(* CODESYS project e!C_ScaleAnalogIO_Test_1.ecp

Project tree, tasks and I/O mapping:
  Device : 750-8202 PFC200 2ETH RS, WAGO, order no. 0750-8202, version 5.11.1.16
    application Application
      libraries: Util, * (System)
      task Test (cyclic, interval T#50ms, priority 11) calls PLC_PRG
      Data types/
      Global Variables/
        global variables Global_Constants
        global variables Global_Retains
        global variables Global_Variables
        global variables Variable_Configuration
      POUs/
        Diagnostic/
          program ModuleDiagnostic [ST]: ModuleDiagList
        Scaling/
          function block fbScale_AI_455 [ST]
          function block fbScale_AI_457 [ST]
          function block fbScale_AI_457_Positiv [ST]
          function block fbScale_AI_460 [ST]
          function block fbScale_AI_461 [ST]
          function block fbScale_AI_466 [ST]
          function block fbScale_AI_473 [ST]
          function block fbScale_AO_552 [ST]
          function block fbScale_AO_555 [ST]
          function block fbScale_AO_556 [ST]
          function block fbScale_AO_559 [ST]
        program PLC_PRG [CFC]: AnalogInput, AnalogOutput
      Visualizations/
      global variables PersistentVars
      trace Sampling_Trace (task ): 
    DeviceAdapter
    Kbus : Kbus, WAGO, version 1.4.0.2
        unmapped channels: K-BUS diagnostics
    MODBUS
      MODBUS : MODBUS, WAGO, order no. n/a, version 1.1.1.15
    Serial
      COM1 : COM1, WAGO, version 0.0.0.19
  GlobalImagePool
*)

// Device/Application/Global Variables/Global_Constants
VAR_GLOBAL CONSTANT

	LIM_OF_DIAG_MODULES : INT := 100;
	LIM_OF_DIAG_CHANNELS : INT := 8;
	MODULE_DIAG_UNDERRANGE : INT := 16#41;
	MODULE_DIAG_OVERRANGE : INT := 16#42;
	MODULE_DIAG_MSG_UNDERRANGE : STRING(15) := 'Underrange';
	MODULE_DIAG_MSG_OVERRANGE : STRING(15) := 'Overrange';
	MODULE_DIAG_MSG_OK : STRING(15) := 'Ok';

END_VAR

// Device/Application/Global Variables/Global_Retains
VAR_GLOBAL RETAIN

	awDiagDataCapture				: ARRAY[1..LIM_OF_DIAG_MODULES, 1..LIM_OF_DIAG_CHANNELS] OF WORD;

END_VAR

// Device/Application/Global Variables/Global_Variables
VAR_GLOBAL

	asModuleDiag				: ARRAY[1..LIM_OF_DIAG_MODULES, 1..LIM_OF_DIAG_CHANNELS] OF STRING(15);

END_VAR

// Device/Application/Global Variables/Variable_Configuration
VAR_CONFIG
END_VAR

// Device/Application/PersistentVars
VAR_GLOBAL PERSISTENT RETAIN
END_VAR

// Device/Application/POUs/PLC_PRG
PROGRAM PLC_PRG
VAR

	Scale_AI_Pressure_1: fbScale_AI_455;
	Scale_AI_Distance_1: fbScale_AI_473;
	Scale_AI_Level_1: fbScale_AI_466;
	Scale_AI_Temp_1: fbScale_AI_460;
	Scale_AI_EngineTemp_1: fbScale_AI_461;
	Scale_AI_SpeedActual_1: fbScale_AI_457_Positiv;
	Scale_AO_SpeedSet_1: fbScale_AO_559;
	Scale_AO_PressureSet_1: fbScale_AO_555;
	Scale_AO_LevelSet_1: fbScale_AO_556;
	Scale_AO_DistanceSet_1: fbScale_AO_552;

	AI_Pressure_1_Signal: REAL;
	AI_Pressure_1_SignalStatus : BYTE;
	AI_Distance_1_Signal: REAL;
	AI_Distance_1_SignalStatus : BYTE;
	AI_Level_1_Signal: REAL;
	AI_Level_1_SignalStatus : BYTE;
	AI_Temp_1_Signal: REAL;
	AI_Temp_1_SignalStatus : BYTE;
	AI_EngineTemp_1_Signal: REAL;
	AI_EngineTemp_1_SignalStatus : BYTE;
	AI_SpeedActual_1_Signal: REAL;
	AI_SpeedActual_1_SignalStatus: BYTE;
	AO_SpeedSet_1_Signal: REAL;
	AO_SpeedSet_1_SignalStatus: BYTE;
	AO_PressureSet_1_Signal: REAL;
	AO_PressureSet_1_SignalStatus: BYTE;
	AO_LevelSet_1_Signal: REAL;
	AO_LevelSet_1_SignalStatus: BYTE;
	AO_DistanceSet_1_Signal: REAL;
	AO_DistanceSet_1_SignalStatus: BYTE;

	AI_455_1_1_sim: WORD;
	AI_473_1_1_sim: WORD;
	AI_466_1_1_sim: WORD;
	AI_460_1_1_sim: INT;
	AI_461_1_1_sim: INT;
	AI_457_1_1_sim: WORD;
	AO_559_1_1_sim: WORD;
	AO_552_1_1_sim: WORD;
	AO_555_1_1_sim: WORD;
	AO_556_1_1_sim: WORD;

END_VAR

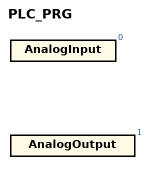
AnalogInput();
AnalogOutput();

ACTION AnalogInput:
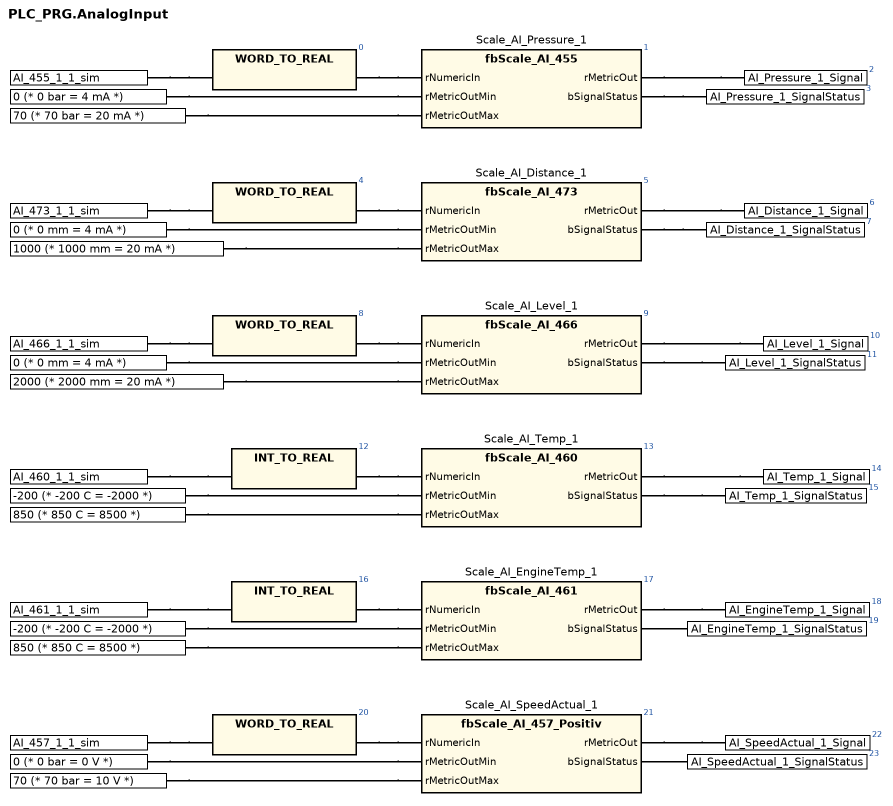
Scale_AI_Pressure_1(
    rNumericIn := WORD_TO_REAL(AI_455_1_1_sim),
    rMetricOutMin := 0 (* 0 bar = 4 mA *),
    rMetricOutMax := 70 (* 70 bar = 20 mA *)); // fbScale_AI_455
AI_Pressure_1_Signal := Scale_AI_Pressure_1.rMetricOut;
AI_Pressure_1_SignalStatus := Scale_AI_Pressure_1.bSignalStatus;
Scale_AI_Distance_1(
    rNumericIn := WORD_TO_REAL(AI_473_1_1_sim),
    rMetricOutMin := 0 (* 0 mm = 4 mA *),
    rMetricOutMax := 1000 (* 1000 mm = 20 mA *)); // fbScale_AI_473
AI_Distance_1_Signal := Scale_AI_Distance_1.rMetricOut;
AI_Distance_1_SignalStatus := Scale_AI_Distance_1.bSignalStatus;
Scale_AI_Level_1(
    rNumericIn := WORD_TO_REAL(AI_466_1_1_sim),
    rMetricOutMin := 0 (* 0 mm = 4 mA *),
    rMetricOutMax := 2000 (* 2000 mm = 20 mA *)); // fbScale_AI_466
AI_Level_1_Signal := Scale_AI_Level_1.rMetricOut;
AI_Level_1_SignalStatus := Scale_AI_Level_1.bSignalStatus;
Scale_AI_Temp_1(
    rNumericIn := INT_TO_REAL(AI_460_1_1_sim),
    rMetricOutMin := -200 (* -200 C = -2000 *),
    rMetricOutMax := 850 (* 850 C = 8500 *)); // fbScale_AI_460
AI_Temp_1_Signal := Scale_AI_Temp_1.rMetricOut;
AI_Temp_1_SignalStatus := Scale_AI_Temp_1.bSignalStatus;
Scale_AI_EngineTemp_1(
    rNumericIn := INT_TO_REAL(AI_461_1_1_sim),
    rMetricOutMin := -200 (* -200 C = -2000 *),
    rMetricOutMax := 850 (* 850 C = 8500 *)); // fbScale_AI_461
AI_EngineTemp_1_Signal := Scale_AI_EngineTemp_1.rMetricOut;
AI_EngineTemp_1_SignalStatus := Scale_AI_EngineTemp_1.bSignalStatus;
Scale_AI_SpeedActual_1(
    rNumericIn := WORD_TO_REAL(AI_457_1_1_sim),
    rMetricOutMin := 0 (* 0 bar = 0 V *),
    rMetricOutMax := 70 (* 70 bar = 10 V *)); // fbScale_AI_457_Positiv
AI_SpeedActual_1_Signal := Scale_AI_SpeedActual_1.rMetricOut;
AI_SpeedActual_1_SignalStatus := Scale_AI_SpeedActual_1.bSignalStatus;
END_ACTION

ACTION AnalogOutput:
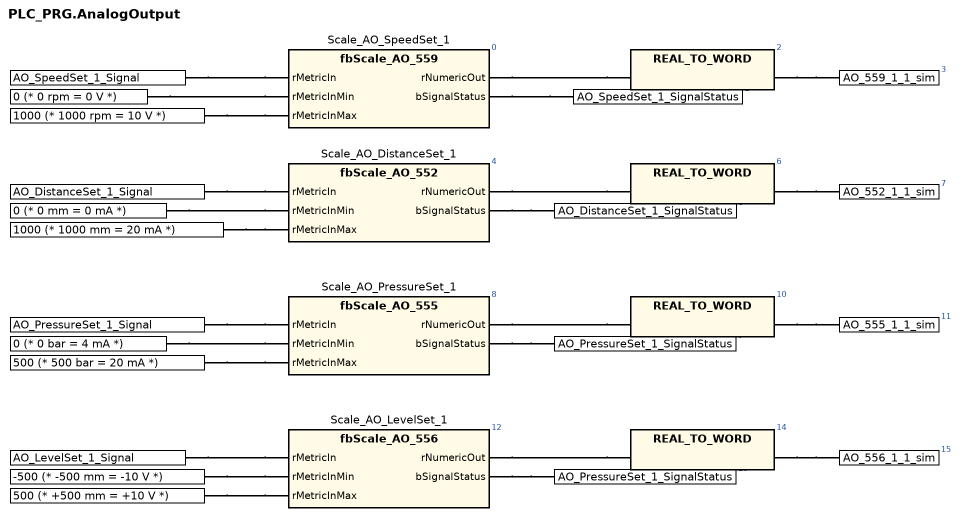
Scale_AO_SpeedSet_1(
    rMetricIn := AO_SpeedSet_1_Signal,
    rMetricInMin := 0 (* 0 rpm = 0 V *),
    rMetricInMax := 1000 (* 1000 rpm = 10 V *)); // fbScale_AO_559
AO_SpeedSet_1_SignalStatus := Scale_AO_SpeedSet_1.bSignalStatus;
AO_559_1_1_sim := REAL_TO_WORD(Scale_AO_SpeedSet_1.rNumericOut);
Scale_AO_DistanceSet_1(
    rMetricIn := AO_DistanceSet_1_Signal,
    rMetricInMin := 0 (* 0 mm = 0 mA *),
    rMetricInMax := 1000 (* 1000 mm = 20 mA *)); // fbScale_AO_552
AO_DistanceSet_1_SignalStatus := Scale_AO_DistanceSet_1.bSignalStatus;
AO_552_1_1_sim := REAL_TO_WORD(Scale_AO_DistanceSet_1.rNumericOut);
Scale_AO_PressureSet_1(
    rMetricIn := AO_PressureSet_1_Signal,
    rMetricInMin := 0 (* 0 bar = 4 mA *),
    rMetricInMax := 500 (* 500 bar = 20 mA *)); // fbScale_AO_555
AO_PressureSet_1_SignalStatus := Scale_AO_PressureSet_1.bSignalStatus;
AO_555_1_1_sim := REAL_TO_WORD(Scale_AO_PressureSet_1.rNumericOut);
Scale_AO_LevelSet_1(
    rMetricIn := AO_LevelSet_1_Signal,
    rMetricInMin := -500 (* -500 mm = -10 V *),
    rMetricInMax := 500 (* +500 mm = +10 V *)); // fbScale_AO_556
AO_PressureSet_1_SignalStatus := Scale_AO_LevelSet_1.bSignalStatus;
AO_556_1_1_sim := REAL_TO_WORD(Scale_AO_LevelSet_1.rNumericOut);
END_ACTION

END_PROGRAM

// Device/Application/POUs/Scaling/fbScale_AI_455
FUNCTION_BLOCK fbScale_AI_455

VAR_INPUT

	rNumericIn: REAL;
	rMetricOutMin: REAL := 4;
	rMetricOutMax: REAL := 20;

END_VAR


VAR_OUTPUT

	rMetricOut: REAL;
	bSignalStatus : BYTE;

END_VAR


VAR

	LIN_TRAFO_ScaleAnalog: LIN_TRAFO;
	rNumericInMin: REAL := 0;
	rNumericInMax: REAL := 32760;

END_VAR



LIN_TRAFO_ScaleAnalog(
	IN			:= rNumericIn,
	IN_MIN		:= rNumericInMin,
	IN_MAX		:= rNumericInMax,
	OUT_MIN		:= rMetricOutMin,
	OUT_MAX		:= rMetricOutMax,
	OUT			=> rMetricOut );


IF ( (REAL_TO_WORD(rNumericIn) AND 16#0003) > 0 ) THEN
	IF (REAL_TO_WORD(rNumericIn) > rNumericInMax) THEN
		rMetricOut := rMetricOutMax;
		bSignalStatus := 2;
	ELSE
		rMetricOut := rMetricOutMin;
		bSignalStatus := 1;
	END_IF
ELSE
	bSignalStatus := 0;
END_IF

END_FUNCTION_BLOCK

// Device/Application/POUs/Scaling/fbScale_AI_473
FUNCTION_BLOCK fbScale_AI_473

VAR_INPUT

	rNumericIn: REAL;
	rMetricOutMin: REAL := 4;
	rMetricOutMax: REAL := 20;

END_VAR


VAR_OUTPUT

	rMetricOut: REAL;
	bSignalStatus : BYTE;

END_VAR


VAR

	LIN_TRAFO_ScaleAnalog: LIN_TRAFO;
	rNumericInMin: REAL := 4096;
	rNumericInMax: REAL := 20480;

END_VAR



LIN_TRAFO_ScaleAnalog(
	IN			:= rNumericIn,
	IN_MIN		:= rNumericInMin,
	IN_MAX		:= rNumericInMax,
	OUT_MIN		:= rMetricOutMin,
	OUT_MAX		:= rMetricOutMax,
	OUT			=> rMetricOut );


IF ( (REAL_TO_WORD(rNumericIn) AND 16#0003) > 0 ) THEN
	IF (REAL_TO_WORD(rNumericIn) > rNumericInMax) THEN
		rMetricOut := rMetricOutMax;
		bSignalStatus := 2;
	ELSE
		rMetricOut := rMetricOutMin;
		bSignalStatus := 1;
	END_IF
ELSE
	bSignalStatus := 0;
END_IF

END_FUNCTION_BLOCK

// Device/Application/POUs/Scaling/fbScale_AI_466
FUNCTION_BLOCK fbScale_AI_466

VAR_INPUT

	rNumericIn: REAL;
	rMetricOutMin: REAL := 4;
	rMetricOutMax: REAL := 20;

END_VAR


VAR_OUTPUT

	rMetricOut: REAL;
	bSignalStatus : BYTE;

END_VAR


VAR

	LIN_TRAFO_ScaleAnalog: LIN_TRAFO;
	rNumericInMin: REAL := 0;
	rNumericInMax: REAL := 32760;

END_VAR



LIN_TRAFO_ScaleAnalog(
	IN			:= rNumericIn,
	IN_MIN		:= rNumericInMin,
	IN_MAX		:= rNumericInMax,
	OUT_MIN		:= rMetricOutMin,
	OUT_MAX		:= rMetricOutMax,
	OUT			=> rMetricOut );


IF ( (REAL_TO_WORD(rNumericIn) AND 16#0003) > 0 ) THEN
	IF (REAL_TO_WORD(rNumericIn) > rNumericInMax) THEN
		rMetricOut := rMetricOutMax;
		bSignalStatus := 2;
	ELSE
		rMetricOut := rMetricOutMin;
		bSignalStatus := 1;
	END_IF
ELSE
	bSignalStatus := 0;
END_IF

END_FUNCTION_BLOCK

// Device/Application/POUs/Scaling/fbScale_AI_460
FUNCTION_BLOCK fbScale_AI_460

VAR_INPUT

	rNumericIn: REAL;
	rMetricOutMin: REAL := -200;
	rMetricOutMax: REAL := 850;

END_VAR


VAR_OUTPUT

	rMetricOut: REAL;
	bSignalStatus : BYTE;

END_VAR


VAR

	LIN_TRAFO_ScaleAnalog: LIN_TRAFO;
	rNumericInMin: REAL := -2000;
	rNumericInMax: REAL := 8500;

END_VAR



LIN_TRAFO_ScaleAnalog(
	IN			:= rNumericIn,
	IN_MIN		:= rNumericInMin,
	IN_MAX		:= rNumericInMax,
	OUT_MIN		:= rMetricOutMin,
	OUT_MAX		:= rMetricOutMax,
	OUT			=> rMetricOut );


IF (rNumericIn >= rNumericInMax) THEN
	rMetricOut := rMetricOutMax;
	bSignalStatus := 1;
ELSIF (rNumericIn < rNumericInMin) THEN
	rMetricOut := rMetricOutMin;
	bSignalStatus := 2;
ELSE
	bSignalStatus := 0;
END_IF

END_FUNCTION_BLOCK

// Device/Application/POUs/Scaling/fbScale_AI_461
FUNCTION_BLOCK fbScale_AI_461

VAR_INPUT

	rNumericIn: REAL;
	rMetricOutMin: REAL := -200;
	rMetricOutMax: REAL := 850;

END_VAR


VAR_OUTPUT

	rMetricOut: REAL;
	bSignalStatus : BYTE;

END_VAR


VAR

	LIN_TRAFO_ScaleAnalog: LIN_TRAFO;
	rNumericInMin: REAL := -2000;
	rNumericInMax: REAL := 8500;

END_VAR



LIN_TRAFO_ScaleAnalog(
	IN			:= rNumericIn,
	IN_MIN		:= rNumericInMin,
	IN_MAX		:= rNumericInMax,
	OUT_MIN		:= rMetricOutMin,
	OUT_MAX		:= rMetricOutMax,
	OUT			=> rMetricOut );


IF (rNumericIn >= rNumericInMax) THEN
	rMetricOut := rMetricOutMax;
	bSignalStatus := 1;
ELSIF (rNumericIn < rNumericInMin) THEN
	rMetricOut := rMetricOutMin;
	bSignalStatus := 2;
ELSE
	bSignalStatus := 0;
END_IF

END_FUNCTION_BLOCK

// Device/Application/POUs/Scaling/fbScale_AI_457_Positiv
FUNCTION_BLOCK fbScale_AI_457_Positiv

VAR_INPUT

	rNumericIn: REAL;
	rMetricOutMin: REAL := -10;
	rMetricOutMax: REAL := 10;

END_VAR


VAR_OUTPUT

	rMetricOut: REAL;
	bSignalStatus : BYTE;

END_VAR


VAR

	LIN_TRAFO_ScaleAnalog: LIN_TRAFO;
	rNumericInMin: REAL := 0;
	rNumericInMax: REAL := 32760;

END_VAR

LIN_TRAFO_ScaleAnalog(
	IN			:= rNumericIn,
	IN_MIN		:= rNumericInMin,
	IN_MAX		:= rNumericInMax,
	OUT_MIN		:= rMetricOutMin,
	OUT_MAX		:= rMetricOutMax,
	OUT			=> rMetricOut );


IF ( (REAL_TO_WORD(rNumericIn) AND 16#0003) > 0 ) THEN
	IF (REAL_TO_WORD(rNumericIn) > rNumericInMax) THEN
		rMetricOut := rMetricOutMax;
		bSignalStatus := 2;
	ELSE
		rMetricOut := rMetricOutMin;
		bSignalStatus := 1;
	END_IF
ELSE
	bSignalStatus := 0;
END_IF

END_FUNCTION_BLOCK

// Device/Application/POUs/Scaling/fbScale_AO_559
FUNCTION_BLOCK fbScale_AO_559

VAR_INPUT

	rMetricIn: REAL;
	rMetricInMin: REAL := 0;
	rMetricInMax: REAL := 10;

END_VAR


VAR_OUTPUT

	rNumericOut: REAL;
	bSignalStatus : BYTE;

END_VAR


VAR

	LIN_TRAFO_ScaleAnalog: LIN_TRAFO;
	rNumericOutMin: REAL := 0;
	rNumericOutMax: REAL := 32767;

END_VAR

LIN_TRAFO_ScaleAnalog(
	IN			:= rMetricIn,
	IN_MIN		:= rMetricInMin,
	IN_MAX		:= rMetricInMax,
	OUT_MIN		:= rNumericOutMin,
	OUT_MAX		:= rNumericOutMax,
	OUT			=> rNumericOut );


IF (rMetricIn > rMetricInMax) THEN
	rNumericOut := rNumericOutMax;
	bSignalStatus := 2;
ELSIF (rMetricIn < rMetricInMin) THEN
	rNumericOut := rNumericOutMin;
	bSignalStatus := 1;
ELSE
	bSignalStatus := 0;
END_IF

END_FUNCTION_BLOCK

// Device/Application/POUs/Scaling/fbScale_AO_555
FUNCTION_BLOCK fbScale_AO_555

VAR_INPUT

	rMetricIn: REAL;
	rMetricInMin: REAL := 4;
	rMetricInMax: REAL := 20;

END_VAR


VAR_OUTPUT

	rNumericOut: REAL;
	bSignalStatus : BYTE;

END_VAR


VAR

	LIN_TRAFO_ScaleAnalog: LIN_TRAFO;
	rNumericOutMin: REAL := 0;
	rNumericOutMax: REAL := 32767;

END_VAR

LIN_TRAFO_ScaleAnalog(
	IN			:= rMetricIn,
	IN_MIN		:= rMetricInMin,
	IN_MAX		:= rMetricInMax,
	OUT_MIN		:= rNumericOutMin,
	OUT_MAX		:= rNumericOutMax,
	OUT			=> rNumericOut );


IF (rMetricIn > rMetricInMax) THEN
	rNumericOut := rNumericOutMax;
	bSignalStatus := 2;
ELSIF (rMetricIn < rMetricInMin) THEN
	rNumericOut := rNumericOutMin;
	bSignalStatus := 1;
ELSE
	bSignalStatus := 0;
END_IF

END_FUNCTION_BLOCK

// Device/Application/POUs/Scaling/fbScale_AO_556
FUNCTION_BLOCK fbScale_AO_556

VAR_INPUT

	rMetricIn: REAL;
	rMetricInMin: REAL := -10;
	rMetricInMax: REAL := 10;

END_VAR


VAR_OUTPUT

	rNumericOut: REAL;
	bSignalStatus : BYTE;

END_VAR


VAR

	LIN_TRAFO_ScaleAnalog: LIN_TRAFO;
	rNumericOutMin: REAL := -32767;
	rNumericOutMax: REAL := 32767;

END_VAR

LIN_TRAFO_ScaleAnalog(
	IN			:= rMetricIn,
	IN_MIN		:= rMetricInMin,
	IN_MAX		:= rMetricInMax,
	OUT_MIN		:= rNumericOutMin,
	OUT_MAX		:= rNumericOutMax,
	OUT			=> rNumericOut );


IF (rMetricIn > rMetricInMax) THEN
	rNumericOut := rNumericOutMax;
	bSignalStatus := 2;
ELSIF (rMetricIn < rMetricInMin) THEN
	rNumericOut := rNumericOutMin;
	bSignalStatus := 1;
ELSE
	bSignalStatus := 0;
END_IF

END_FUNCTION_BLOCK

// Device/Application/POUs/Scaling/fbScale_AO_552
FUNCTION_BLOCK fbScale_AO_552

VAR_INPUT

	rMetricIn: REAL;
	rMetricInMin: REAL := 0;
	rMetricInMax: REAL := 20;

END_VAR


VAR_OUTPUT

	rNumericOut: REAL;
	bSignalStatus : BYTE;

END_VAR


VAR

	LIN_TRAFO_ScaleAnalog: LIN_TRAFO;
	rNumericOutMin: REAL := 0;
	rNumericOutMax: REAL := 32767;

END_VAR

LIN_TRAFO_ScaleAnalog(
	IN			:= rMetricIn,
	IN_MIN		:= rMetricInMin,
	IN_MAX		:= rMetricInMax,
	OUT_MIN		:= rNumericOutMin,
	OUT_MAX		:= rNumericOutMax,
	OUT			=> rNumericOut );


IF (rMetricIn > rMetricInMax) THEN
	rNumericOut := rNumericOutMax;
	bSignalStatus := 2;
ELSIF (rMetricIn < rMetricInMin) THEN
	rNumericOut := rNumericOutMin;
	bSignalStatus := 1;
ELSE
	bSignalStatus := 0;
END_IF

END_FUNCTION_BLOCK

// Device/Application/POUs/Diagnostic/ModuleDiagnostic
PROGRAM ModuleDiagnostic
VAR
(*
	GET_TERMINALDIAG : GET_TERMINALDIAG;
	EN : BOOL := TRUE;
	ENO:BOOL;
	TERMINAL:WORD;
	CHANNEL:WORD;
	DIAGDATA:WORD;
	TON_DiagInterval: TON;
	tDiagInterval: TIME := T#200ms;
*)
	iModuleNumber: INT;
	iChannelNumber: INT;
END_VAR



;
(*
GET_TERMINALDIAG(
	EN			:= EN,
	ENO			=> ENO,
	TERMINAL	=> TERMINAL,
	CHANNEL		=> CHANNEL,
	DIAGDATA	=> DIAGDATA);

IF (ENO = TRUE) THEN
	EN := FALSE;
	IF (TERMINAL <> 0) THEN
		awDiagDataCapture[TERMINAL,CHANNEL] := DIAGDATA;
	END_IF
ELSE
	IF (EN = FALSE) THEN
		TON_DiagInterval(IN:= TRUE, PT:= tDiagInterval);
		IF (TON_DiagInterval.Q = TRUE) THEN
			TON_DiagInterval(IN:= FALSE);
			EN := TRUE;
		END_IF
	END_IF
END_IF

ModuleDiagList();
*)

ACTION ModuleDiagList:

FOR iModuleNumber := 1 TO LIM_OF_DIAG_MODULES DO
	FOR iChannelNumber := 1 TO LIM_OF_DIAG_CHANNELS DO
		IF (awDiagDataCapture[iModuleNumber,iChannelNumber] = MODULE_DIAG_UNDERRANGE) THEN
			asModuleDiag[iModuleNumber,iChannelNumber] := MODULE_DIAG_MSG_UNDERRANGE;
		ELSIF (awDiagDataCapture[iModuleNumber,iChannelNumber] = MODULE_DIAG_OVERRANGE) THEN
			asModuleDiag[iModuleNumber,iChannelNumber] := MODULE_DIAG_MSG_OVERRANGE;
		ELSE
			asModuleDiag[iModuleNumber,iChannelNumber] := MODULE_DIAG_MSG_OK;
		END_IF
	END_FOR
END_FOR
END_ACTION

END_PROGRAM

// Device/Application/POUs/Scaling/fbScale_AI_457
FUNCTION_BLOCK fbScale_AI_457

VAR_INPUT

	rNumericIn: REAL;
	rMetricOutMin: REAL := -10;
	rMetricOutMax: REAL := 10;

END_VAR


VAR_OUTPUT

	rMetricOut: REAL;
	bSignalStatus : BYTE;

END_VAR


VAR

	LIN_TRAFO_ScaleAnalog: LIN_TRAFO;
	rNumericInMin: REAL := -32768;
	rNumericInMax: REAL := 32760;

END_VAR

LIN_TRAFO_ScaleAnalog(
	IN			:= rNumericIn,
	IN_MIN		:= rNumericInMin,
	IN_MAX		:= rNumericInMax,
	OUT_MIN		:= rMetricOutMin,
	OUT_MAX		:= rMetricOutMax,
	OUT			=> rMetricOut );


IF ( (REAL_TO_WORD(rNumericIn) AND 16#0003) > 0 ) THEN
	IF (REAL_TO_WORD(rNumericIn) > rNumericInMax) THEN
		rMetricOut := rMetricOutMax;
		bSignalStatus := 2;
	ELSE
		rMetricOut := rMetricOutMin;
		bSignalStatus := 1;
	END_IF
ELSE
	bSignalStatus := 0;
END_IF

END_FUNCTION_BLOCK
